# B&R Automation Studio project QuickGate
Automation Studio 4.7.3.93 SP

## Configuration MainPrototype

CPU X20CP0411, AutomationRuntime A4.73, Build 4.1.2, Vc V4.72.0

### Task classes (Cpu.sw)
```
Cyclic#4 (cycle 100000 us, tolerance 100000 us):
  MotorContr <- MotorControl.prg
```

### Hardware
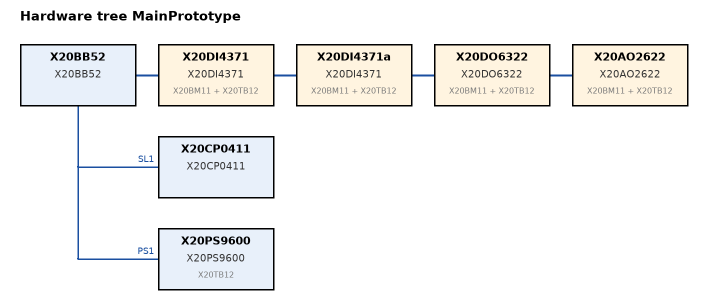
```
X20AO2622 : X20AO2622 v1.1.0.0  [SS1 -> X20TB12c.SS; SL -> X20BM11b.SL1]
X20BB52 : X20BB52 v1.1.0.0
X20BM11 : X20BM11 v1.0.0.1  [X2X1 -> X20BB52.IF6]
X20BM11a : X20BM11 v1.0.0.1  [X2X1 -> X20BM11c.X2X2]
X20BM11b : X20BM11 v1.0.0.1  [X2X1 -> X20BM11a.X2X2]
X20BM11c : X20BM11 v1.0.0.1  [X2X1 -> X20BM11.X2X2]
X20CP0411 : X20CP0411 v1.2.1.0  [SL -> X20BB52.SL1]
  Connector IF2:
    ActivateDevice = 1
    Mode = DHCP Server
    InternetAddress = 169.254.39.254
  ConfigurationID = QuickGate_Config1
  TimerDeviceType = SWIOTIMER
  Cyclic1Duration = 10000
  Cyclic1Tolerance = 10000
  Cyclic2Duration = 20000
  Cyclic2Tolerance = 20000
  Cyclic3Duration = 50000
  Cyclic3Tolerance = 50000
  Cyclic4Duration = 100000
  Cyclic4Tolerance = 100000
  Cyclic5Duration = 200000
  Cyclic5Tolerance = 200000
  Cyclic6Duration = 500000
  Cyclic6Tolerance = 500000
  Cyclic7Duration = 1000000
  Cyclic7Tolerance = 1000000
  Cyclic8Duration = 10000
  Cyclic8Tolerance = 30000000
X20DI4371 : X20DI4371 v1.0.3.0  [SS1 -> X20TB12a.SS; SL -> X20BM11.SL1]
X20DI4371a : X20DI4371 v1.0.3.0  [SS1 -> X20TB12d.SS; SL -> X20BM11c.SL1]
X20DO6322 : X20DO6322 v1.0.4.0  [SS1 -> X20TB12b.SS; SL -> X20BM11a.SL1]
X20PS9600 : X20PS9600 v1.0.1.0  [PS -> X20BB52.PS1; SS1 -> X20TB12.SS]
X20TB12 : X20TB12 v1.0.0.0
X20TB12a : X20TB12 v1.0.0.0
X20TB12b : X20TB12 v1.0.0.0
X20TB12c : X20TB12 v1.0.0.0
X20TB12d : X20TB12 v1.0.0.0
```

### IoMap.iom - X20CP0411/IoMap.iom
```iecst
VAR_CONFIG
	::MotorContr:io.motor.Start_Stop AT %QX."X20DO6322".DigitalOutput01;
	::MotorContr:io.motor.Run_Brake AT %QX."X20DO6322".DigitalOutput02;
	::MotorContr:io.motor.CW_CCW AT %QX."X20DO6322".DigitalOutput03;
	::MotorContr:io.motor.Speed AT %QW."X20AO2622".AnalogOutput01;
	::MotorContr:io.di_tapeswitchYellow AT %IX."X20DI4371".DigitalInput01;
	::MotorContr:io.di_tapeswitchBlack AT %IX."X20DI4371".DigitalInput02;
	::MotorContr:io.di_forwardButton AT %IX."X20DI4371".DigitalInput03;
	::MotorContr:io.di_backwardButton AT %IX."X20DI4371".DigitalInput04;
	::MotorContr:io.di_limitBottom AT %IX."X20DI4371a".DigitalInput01;
	::MotorContr:io.di_limitTop AT %IX."X20DI4371a".DigitalInput02;
END_VAR
```

## Logical view

### Program Logical/MotorControl (IEC)

#### Types.typ
```iecst
TYPE
	io_type : 	STRUCT
		motor : motor_type;
		di_limitBottom : BOOL;
		di_limitTop : BOOL;
		di_tapeswitchBlack : BOOL;
		di_tapeswitchYellow : BOOL;
		di_forwardButton : BOOL;
		di_backwardButton : BOOL;
	END_STRUCT;
	motor_type : 	STRUCT  (*TRUE_FALSE*)
		Run_Brake : BOOL; (*TRUE_FALSE
*)
		CW_CCW : BOOL; (*TRUE_FALSE
*)
		Start_Stop : BOOL; (*TRUE_FALSE
*)
		Speed : INT;
	END_STRUCT;
	Direction_Type : 	STRUCT
	END_STRUCT;
END_TYPE
```

#### Variables.var
```iecst
VAR
	io : io_type;
END_VAR
```

#### Main.st
```iecst
PROGRAM _INIT
	io.motor.Speed := 5000;

END_PROGRAM

PROGRAM _CYCLIC
	(* Insert code here *)
	IF io.di_tapeswitchBlack OR io.di_tapeswitchYellow THEN
		io.motor.Run_Brake := FALSE;
	ELSIF EDGEPOS (io.di_backwardButton) OR EDGEPOS (io.di_forwardButton) THEN
		io.motor.Run_Brake := TRUE;
	END_IF;

	IF io.di_forwardButton THEN
		io.motor.CW_CCW := TRUE;
		io.motor.Start_Stop := TRUE;

	ELSIF io.di_backwardButton THEN
		io.motor.CW_CCW := FALSE;
		io.motor.Start_Stop := TRUE;

	ELSE
		io.motor.Start_Stop := FALSE;
	END_IF;

	IF NOT io.di_limitBottom OR NOT io.di_limitTop THEN
		io.motor.Start_Stop := FALSE;
	END_IF

END_PROGRAM

PROGRAM _EXIT
	(* Insert code here *)

END_PROGRAM
```

Listed in the project but not available here: Logical/Global.typ, Logical/Global.var, Logical/Libraries
